(* CoDeSys 2.3.9.50 project: 6E.pr6 *)
(* Libraries: STANDARD.LB6 5.6.98 12:03:02 *)

(* POU MAIN, LD *)
PROGRAM MAIN
VAR
	CountIncrease AT %IX0.0: BOOL;
	Registervalue: CTU;
	reset AT %IX0.7: BOOL;
	OR005 AT %QX0.0: BOOL;
	OR000 AT %QX0.1: BOOL;
	OR002 AT %QX0.2: BOOL;
END_VAR
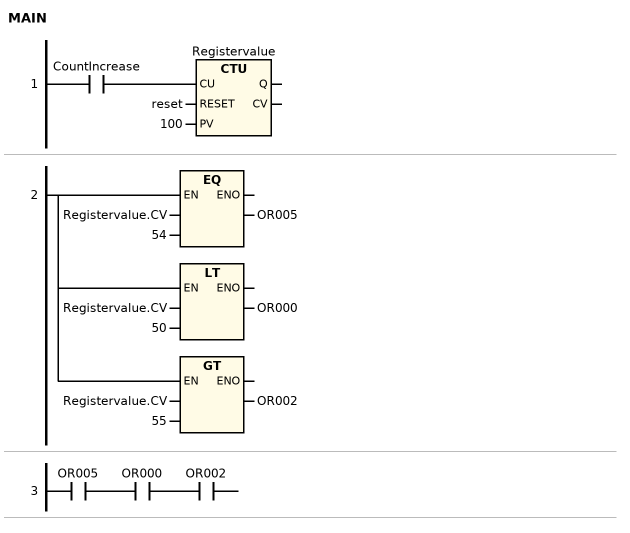
_LD_ (* Ladder Diagram *)
NETWORK 1
	[CountIncrease] - Registervalue:CTU(CU: *, RESET: reset, PV: 100)
NETWORK 2
	*
		EN --- EQ(Registervalue.CV, 54) => OR005
		EN --- LT(Registervalue.CV, 50) => OR000
		EN --- GT(Registervalue.CV, 55) => OR002
NETWORK 3
	[OR005] - [OR000] - [OR002]
_END_LD_
(* the same logic as Structured Text *)
(* Network 1 *)
Registervalue(CU := CountIncrease, RESET := reset, PV := 100);
(* Network 2 *)
OR005 := Registervalue.CV = 54;
OR000 := Registervalue.CV < 50;
OR002 := Registervalue.CV > 55;
(* Network 3 *)
END_PROGRAM
